Fanuc KAREL source: kd00066.KL

-- PROVISIONAL review KL for V770-1; original PC SHA256 4ec88c306d501eea202a1bbcb4c2830faa65225685b553a4d96ee1a20cf40acf
-- Incomplete behavior may be omitted. Consult companion uncertainty JSON. Do not deploy.
PROGRAM KD00066
%NOLOCKGROUP
VAR
  I : INTEGER
  J : INTEGER
  B : BOOLEAN
  R : REAL
  S : STRING[80]
BEGIN
  -- UNRESOLVED_PC offsets 5-17; opcodes 9D,81,18,9D,1B,9D,12,13,04
  -- UNRESOLVED_PC offsets 22-26; opcodes 7F
END KD00066
